// Function block to control simple MCC 
FUNCTION_BLOCK FB_MotorControl
VAR
	autoButton		    : Button;	// Scada Button auto
	forwardButton		: Button;	// Scada Button forward

	
	iDrive 		: I_Drive;				// interface variable
	eStateDevice : E_StateDevice;     // text information about drive 'OFF', 'ON', 'FAULT', 'RUNNING'
	
END_VAR

// Check the Drive status
eStateDevice := iDrive.StatusState();



//Button Auto is set in SCADA motor control station, but Client in PLC have to have acces too directly via a variable to work in Auto mode
IF autoButton.IsPressed THEN 
	AutoOn();	// Turn On SCADA auto Led
ELSE
	AutoOff(); // Turn Off SCADA auto Led
	
	// IF NOT AUTO MODE THEN, EXECUTE
	
	CASE eStateDevice OF
		eOn :
			 IF forwardButton.IsPressed THEN
				ForwardOn();
			 END_IF
				 
		eOff :
			ForwardOff();
			iDrive.WorkCounterOff();
				
		eForward :
			IF forwardButton.IsPressed THEN
				iDrive.WorkCounterOn();
            	iDrive.WorkCount();			
			ELSE	
				ForwardOff();
				iDrive.WorkCounterOff();
			 END_IF
		
		eFault :
			iDrive.WorkCounterOff();
	
	END_CASE

END_IF

METHOD PUBLIC AutoOff : BOOL
VAR_INPUT
END_VAR
iDrive.AutoLedOff();
END_METHOD

METHOD PUBLIC AutoOn : BOOL
VAR_INPUT
END_VAR
iDrive.AutoLedOn();
END_METHOD

METHOD FB_init : BOOL
VAR_INPUT
	bInitRetains : BOOL; // if TRUE, the retain variables are initialized (warm start / cold start)
	bInCopyCode  : BOOL;  // if TRUE, the instance afterwards gets moved into the copy code (online change)
	iDrive		 : I_Drive;
END_VAR
THIS^.iDrive := iDrive;
END_METHOD

METHOD PUBLIC ForwardOff : BOOL
VAR_INPUT

END_VAR
ForwardOff := iDrive.SwitchOff();
END_METHOD

METHOD PUBLIC ForwardOn : BOOL
VAR_INPUT

END_VAR
ForwardOn := iDrive.SwitchOn();
END_METHOD

END_FUNCTION_BLOCK

(* stored: Version 1.1.0.1, ProductVersion 3.1.4024.12
   POU FB_MotorControl: Id {cb429039-0c12-4649-8c7a-84a654602980}, SpecialFunc None
   Method AutoOff: Id {d8967504-f11e-4755-939d-967045b0616b}
   Method AutoOn: Id {28b9c243-c4ee-4cbe-83aa-fef6a3c2a841}
   Method FB_init: Id {30ce9704-a946-441a-bf51-690ce8812f28}
   Method ForwardOff: Id {fc03a760-fdef-4db9-b431-c6ea7e47b138}
   Method ForwardOn: Id {ebe68f71-77b6-4a31-b726-f94b2b996811} *)
